# EPICS StreamDevice protocol: fimscbApp/Db/stream_raw.proto
sendRawCommand {
  out "%s";
}

sendRawQuery {
  ExtraInput = Ignore;
  out "%s";
  in  "%(\$1)40c";
}
